{attribute addProperty BoxType "EK1122-0000-0018"}
{attribute addProperty Id "Beckhoff_EL3xxxsub_EK1100EK1100_179A0949162"}
{attribute addProperty CRC "2682426131"}
{attribute addProperty SizeInBites "16"}
{attribute addProperty SizeInBytes "2"}
TYPE Beckhoff_EL3xxxEK1122_9FE29313 EXTENDS EK1122_179A0949 :
STRUCT
	{attribute addProperty Name "Beckhoff_EL3xxxsub_EK1100"}
	Beckhoff_EL3xxxsub_EK1100 : EK1100_179A0949;
END_STRUCT
END_TYPE

(* stored: Version 1.2.0.0, ProductVersion 3.1.4024.9
   DUT Beckhoff_EL3xxxEK1122_9FE29313: Id {711af001-b7c4-472b-a6d0-99cff42c9786} *)
